// TIA Portal V19 export
VAR_GLOBAL   // PLC tag table "D22"
   D22_Lp_EntryReq_LB305 AT %Q300.0 : Bool;   // 268SH1
   D22_Lp_EntryReq_LB306 AT %Q350.0 : Bool;   // 269SH1
   D22_Lp_SafetyReset_LB305 AT %Q300.1 : Bool;   // 268SH2
   D22_Lp_SafetyReset_LB306 AT %Q350.1 : Bool;   // 269SH2
   D22_Pb_EntryReq_LB305 AT %I300.3 : Bool;   // 268SH1
   D22_Pb_EntryReq_LB306 AT %I350.0 : Bool;   // 269SH1
   D22_Pb_SafetyReset_LB305 AT %I300.4 : Bool;   // 268SH2
   D22_Pb_SafetyReset_LB306 AT %I350.1 : Bool;   // 269SH2
   D22_Ls AT %I1400.2 : Bool;   // 300DI2 - 268BE1/R1
END_VAR
